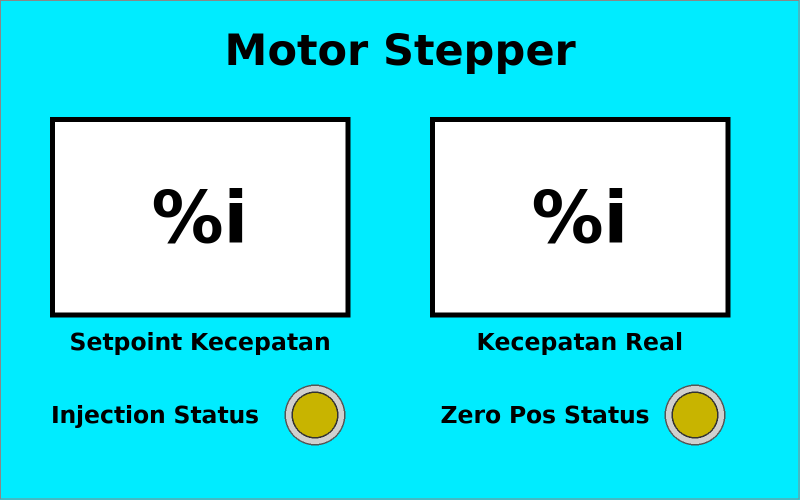
VISUALIZATION Screen_2_Sub_5  // 800x500
    Rectangle (0,0 800x500)
    Label (0,0 800x100), "Motor Stepper"
    Rectangle (50,117 300x200), "%i", text variable: GVL.HMI_Motor_Stepper_Input
        OnMouseClick: write GVL.HMI_Motor_Stepper_Input via VisuDialogs.Numpad
    Label (50,317 300x50), "Setpoint Kecepatan"
    Label (430,317 300x50), "Kecepatan Real"
    Rectangle (430,117 300x200), "%i", text variable: GVL.HMI_Motor_Stepper_Real
    Lamp1 (280,380 70x70), variable: GVL.HMI_Motor_Stepper_Injec_Stat, style: Lamp-Lamp1-Yellow
    Lamp1 (660,380 70x70), variable: GVL.HMI_Motor_Stepper_Zero_Pos, style: Lamp-Lamp1-Yellow
    Label (35,390 240x50), "Injection Status"
    Label (425,390 240x50), "Zero Pos Status"
END_VISUALIZATION

(* stored: Version 1.1.0.1, ProductVersion 3.1.4024.12
   Visu Screen_2_Sub_5: Id {baa82643-73e1-4b36-8463-6245669ff660} *)
